// TIA Portal V18 export
FUNCTION "mot_speed_blind" : Void   // FC11, FBD
{ S7_Optimized_Access := 'TRUE' }
VERSION : 0.1
// stored: AutoNumber true, IsIECCheckEnabled false, SetENOAutomatically false, UDAEnableTagReadback false
   VAR_INPUT
      SET_SPEED : Real;
      par_speed_blind : Real;
      xFwdOK : Bool;
      xRevOK : Bool;
   END_VAR
   VAR_OUTPUT
      speed_calculated : Real;
   END_VAR
   VAR_TEMP
      go_fwd : Bool;
      go_rev : Bool;
   END_VAR
BEGIN

REGION Network 1
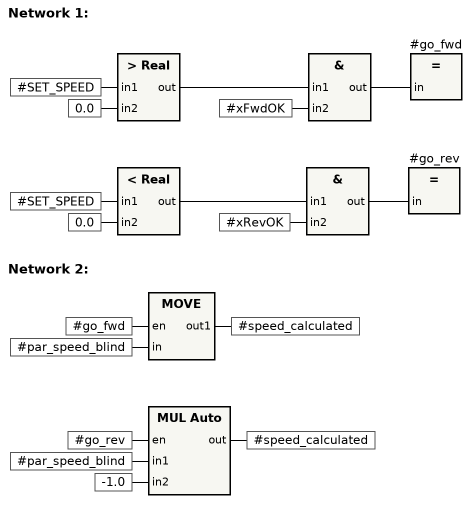
   #go_fwd := (#SET_SPEED > 0.0) AND #xFwdOK;
   #go_rev := (#SET_SPEED < 0.0) AND #xRevOK;
END_REGION

REGION Network 2
   IF #go_fwd THEN #speed_calculated := #par_speed_blind; END_IF;
   IF #go_rev THEN #speed_calculated := #par_speed_blind * (-1.0); END_IF;
END_REGION
END_FUNCTION
